PROGRAM PRG_08_AutoCrossCut
VAR
	iStep: INT;
	TON_DownDelay: TON;
	ctu_DoublePass: CTU;
	bDoublePassCountUp: BOOL;
	bAutoUp: BOOL;
	bAutoDown: BOOL;
	bAutoCut: BOOL;
	bAutoReturn: BOOL;
	TON_bAutoUp: TON;
	bTON_AutoUp: BOOL;
	R_TRIG_0: R_TRIG;
	TON_AutoCrossCutError: TON;
	SR_DoublePass: SR;
	bDoublePassQ: BOOL;
END_VAR

	IF		NOT bSafetyOK OR IN_FaultReset OR NOT OUT_bSawON OR bAnyServoError
	THEN	iStep	:=	0;
	END_IF

	TON_DownDelay(IN:= , PT:= T#3S, Q=> , ET=> );
	IF		iStep <> 30 THEN
			TON_DownDelay.IN	:= FALSE ;
	END_IF
(* Double Pass counter BOOL *)
	IF		ctu_DoublePass.CV	=	1
	THEN	bDoublePassCountUp		:=	TRUE;
	ELSE	bDoublePassCountUp		:=	FALSE;
	END_IF

CASE iStep OF 
	0:		//	Step 0	:	Init step
				bAutoCrossCut	:= FALSE ;
				bAutoUp			:= FALSE ;
				bAutoDown		:= FALSE ;
				bAutoCut		:= FALSE ;
				bAutoReturn		:= FALSE ;
				bTON_AutoUp		:= FALSE ;
				
		IF
				bSafetyOK
				AND bTurret045Range
				AND OUT_bSawON
				AND (bAutoCrossCutReady AND IN_bAutoCrossCut AND NOT bRemote)
				AND NOT bMachineHoming
				AND NOT bCarriageCentreReference
		THEN
				bAutoCrossCut := TRUE	;
				iStep	:=		20		;
		ELSE
				bAutoCrossCut := FALSE	;
				iStep	:=		0		;
		END_IF

	20:		// Step 20	:	Saw RETURN movement
		IF 
				bAutoCrossCut
				AND bSafetyOK
				AND NOT bLimitRight
			
		THEN	bAutoReturn	:=	TRUE	;
		
		ELSE
				bAutoReturn	:=	FALSE	;
				iStep		:=	30		;
		END_IF
	
		IF 		NOT bSafetyOK
		THEN 	
				bAutoReturn	:=	FALSE	;
				iStep		:=	0		;
		END_IF
		
	30:		// Step 30	:	Saw DOWN movement
	ctu_DoublePass.CV;
		IF
				bAutoCrossCut
				AND bSafetyOK
				AND ((bAutoCrossCutDouble (*AND IN_bDoublePassReference*) AND bDoublePassCountUp) 
					OR ( IN_bDownLimit AND (bDoublePassQ OR NOT bDoublePassCountUp)))
		THEN	
				bAutoDown	:=	TRUE	;
		ELSE
				bAutoDown	:=	FALSE	;
				TON_DownDelay.IN := TRUE ;
					IF TON_DownDelay.Q THEN
						iStep	:=	40		;
					END_IF
		END_IF
		
		IF 		NOT bSafetyOK
		THEN 	
				bAutoDown	:=	FALSE	;
				iStep		:=	0		;
		END_IF
	
	40:		// Step 40	:	Saw CUT movement
		IF
				bAutoCrossCut
				AND bSafetyOK
				AND	NOT bLimitLeft
			THEN
				bAutoCut	:=	TRUE	;
		ELSE
				bAutoCut	:=	FALSE	;
				iStep		:=	50		;
		END_IF
		
		IF 		NOT bSafetyOK
			THEN 	
				bAutoCut	:=	FALSE	;
				iStep		:=	0		;
		END_IF
	
	50:		// Step 50	:	Saw UP movement		(* for double pass: only lift slightly, RETURN, then plunge all the way down *)
	ctu_DoublePass.CV;	
		IF
				bAutoCrossCutDouble AND bDoublePassCountUp AND NOT bDoublePassQ
			THEN
				bTON_AutoUp	:=	TRUE	;
				bAutoUp		:=	NOT TON_bAutoUp.Q	;
				
				IF
					R_TRIG_0.Q THEN
					iStep	:=	60	;
				END_IF
				
		ELSIF
				bAutoCrossCut
				AND bSafetyOK
				AND bSawUpLimit
				AND ((bDoublePassQ AND NOT bDoublePassCountUp AND bAutoCrossCutDouble) OR (NOT bAutoCrossCutDouble))
			THEN
				bAutoUp		:=	TRUE	;
		ELSE
				bAutoUp		:=	FALSE	;
				iStep		:=	60		;
		END_IF
		
		IF 		NOT bSafetyOK
		THEN 	
				bAutoUp		:=	FALSE	;
				iStep		:=	0		;
		END_IF
	
	60:		// Step 60	:	Saw RETURN movement (loop back to step 20 if double pass)
		IF
				bAutoCrossCutDouble
				AND bDoublePassCountUp
		THEN
				iStep		:=	20		;
		ELSIF	
				bAutoCrossCut
				AND bSafetyOK
				AND NOT bCrossCutCentre
		THEN
				bAutoReturn	:=	TRUE	;
		ELSE
				bAutoReturn	:=	FALSE	;
				iStep		:=	0		;
		END_IF
	
END_CASE

ACTION ACT_08_1_AutoCrossCut:
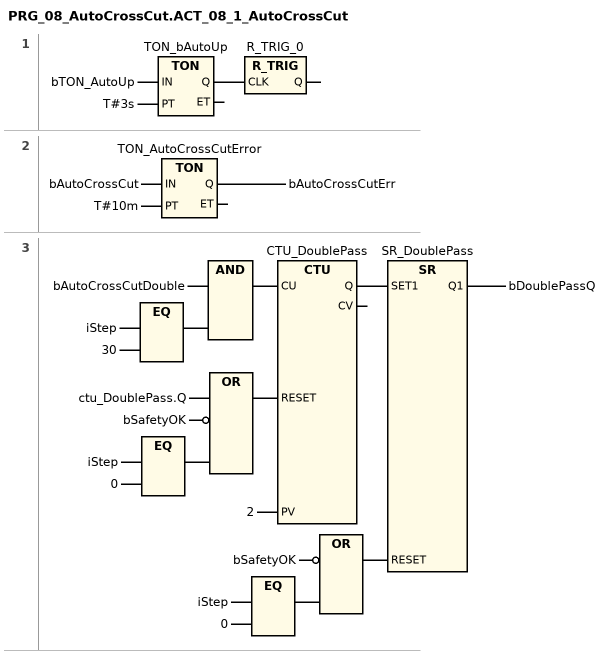
// NETWORK 1
TON_bAutoUp(IN := bTON_AutoUp, PT := T#3s); // TON
R_TRIG_0(CLK := TON_bAutoUp.Q); // R_TRIG

// NETWORK 2
TON_AutoCrossCutError(IN := bAutoCrossCut, PT := T#10m); // TON
bAutoCrossCutErr := TON_AutoCrossCutError.Q;

// NETWORK 3
CTU_DoublePass(
    CU := bAutoCrossCutDouble AND iStep = 30,
    RESET := ctu_DoublePass.Q OR NOT bSafetyOK OR iStep = 0,
    PV := 2); // CTU
SR_DoublePass(SET1 := CTU_DoublePass.Q, RESET := NOT bSafetyOK OR iStep = 0); // SR
bDoublePassQ := SR_DoublePass.Q1;
END_ACTION

END_PROGRAM

(* stored: Version 1.1.0.1, ProductVersion 3.1.4024.15
   POU PRG_08_AutoCrossCut: Id {73f4070d-b53d-44b0-b7c0-d862c4fca4a8}, SpecialFunc None
   Action ACT_08_1_AutoCrossCut: Id {63a0db5e-5485-4feb-b0e7-b93f232749ba} *)
